RoboDK station: 로봇팔 이동.rdk

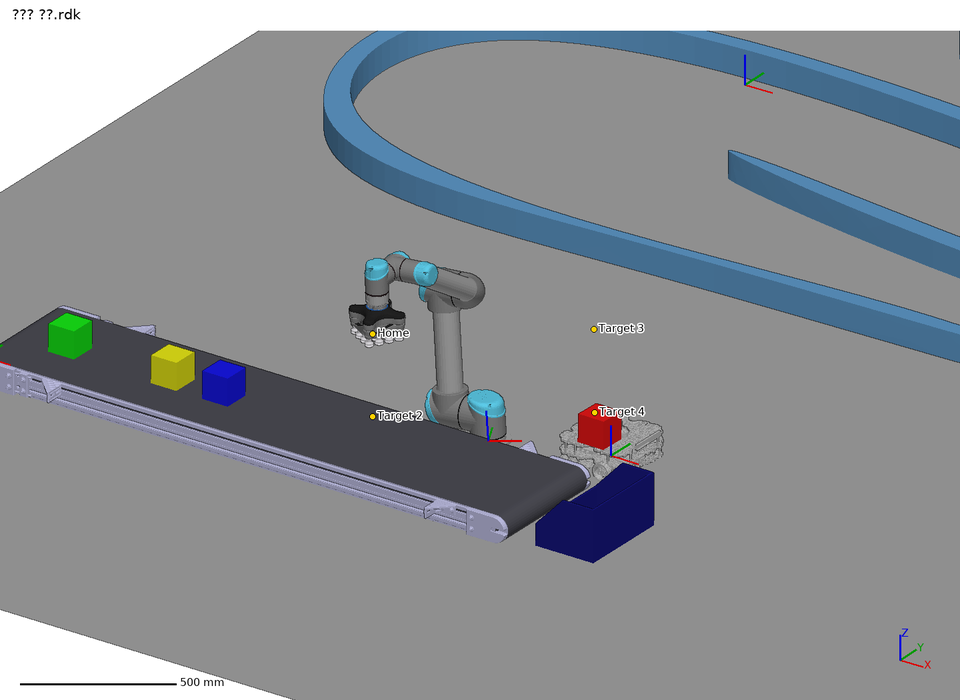
[picture v0: the station drawn from its stored meshes, robots at their saved joint values, targets as dots, program paths as lines]
Station 로봇팔 이동 (saved by RoboDK 5.7.4). Poses are relative to the parent item; angles as X-Y-Z fixed-axis rotations.
Station parameters (name, value as stored): LOAD_READY, 1
  - frame MainFrame at (0, 0, 0) mm
    - target Home (Cartesian target) at (651.26, -3006.26, 497.49) mm, rotated rx -179.45 ry 0.15 rz -30.37 deg; joints [-119.255, -87.831, -60.137, -122.512, 86.049, -150.839] of UR5
    - target Target 2 (Cartesian target) at (637.94, -2986.86, 192) mm, rotated rx -178.43 ry 0.43 rz -30.31 deg; joints [-119.878, -81.815, -111.866, -77.787, 86.288, -151.442] of UR5
    - target Target 3 (Cartesian target) at (1212.52, -2572.15, 497.3) mm, rotated rx -179.45 ry 0.15 rz -30.37 deg; joints [-13.799, -91.747, -62.441, -119.492, 91.513, -45.448] of UR5
    - target Target 4 (Cartesian target) at (1213.24, -2569.51, 200.09) mm, rotated rx -179.45 ry 0.15 rz -30.37 deg; joints [-12.8, -86.409, -112.222, -75.023, 91.577, -44.451] of UR5
  - frame UR5 Base at (820, -2600, 0) mm, rotated rx -1.94 ry -3.6 rz 28.07 deg
    - robot UR5: 6 axes
        modified DH rows (alpha deg, a mm, theta deg, d mm): 0, 0, 0, 89.2; 90, 0, 180, 0; 0, 425, 0, 0; 0, 392, 0, 109.3; -90, 0, 0, 94.75; 90, 0, 180, 82.5
        joint limits [-360, -360, -360, -360, -360, -360] to [360, 360, 360, 360, 360, 360]; home [0, -90, -90, 0, 90, 0]; saved at [-114.958, -89.114, -59.218, -122.443, 86.096, -146.532]
      - tool OnRobot VG10 Vacuum Gripper, TCP at (-36.63, 0, 130.9) mm, size 145.4 x 145.4 x 118.3 mm
  - object Floor at (0, -3000, 0) mm, size 3000 x 3000 x 0 mm, geometry from Floor (1).sld
  - object Floor at (3000, -3000, 0) mm, size 3000 x 3000 x 0 mm, geometry from Floor (1).sld
  - object Floor at (0, 0, 0) mm, size 3000 x 3000 x 0 mm, geometry from Floor (1).sld
  - object Bin Red at (2930, 150, 0) mm, rotated rx 0 ry 0 rz -180 deg, size 225 x 337.5 x 191.2 mm, geometry from Bin-Red.sld
  - object Floor at (3000, 0, 0) mm, size 3000 x 3000 x 0 mm, geometry from Floor (1).sld
  - object Bin Blue at (1380, -2800, 0) mm, rotated rx 0 ry 0 rz -180 deg, size 225 x 337.5 x 191.2 mm, geometry from Bin-Blue.sld
  - object path at (5000, -200, 0) mm, size 3159.6 x 1446.5 x 100 mm, geometry from path.step
  - object path2 at (-2520, -560, 40) mm, rotated rx 0 ry 0 rz 180 deg, size 3159.6 x 1446.5 x 100 mm, geometry from path.step
  - frame Conveyor Belt (2m) Base at (-740, -3190, 100) mm
    - robot Conveyor Belt (2m): 1 axes
        modified DH rows (alpha deg, a mm, theta deg, d mm): 0, 0, 0, 0 linear
        base shift (0, 0, 0) mm, rotated rx 0 ry 90 rz 0 deg
        joint limits [-500000] to [500000]; home [0]; saved at [0]
    - object Blue at (800, 200, 0) mm, size 100 x 100 x 100 mm, geometry from Blue.step
    - object Yellow at (600, 200, 0) mm, size 100 x 100 x 100 mm, geometry from Yellow.step
    - object Green at (200, 200, 0) mm, size 100 x 100 x 100 mm, geometry from Green.step
  - frame turtlebot Base at (1224.75, -2495.03, 20) mm
    - object turtlebot3_waffle (1) at (0, 0, 0) mm, size 280.7 x 305.1 x 138.1 mm, geometry from turtlebot3_waffle (1).step
    - object Red at (10.09, -79.28, 88.06) mm, rotated rx -1.02 ry 0.28 rz -0.1 deg, size 100 x 100 x 100 mm, geometry from Red.step
  - Python program Prog1 (listed below)

--- Python program Prog1 ---
from robodk import robolink
import time

RDK = robolink.Robolink()

# =========================
# RoboDK 아이템 찾기
# =========================
robot = RDK.Item("UR5")
tool = RDK.Item("OnRobot VG10 Vacuum Gripper")
red_box = RDK.Item("Red")
turtle_base = RDK.Item("turtlebot Base")

home = RDK.Item("Home")
target2 = RDK.Item("Target 2")   # Pick 위치
target3 = RDK.Item("Target 3")   # 이동 중간 위치
target4 = RDK.Item("Target 4")   # Place 위치

def check(item, name):
    if not item.Valid():
        raise Exception(f"'{name}' 을 찾을 수 없습니다. 왼쪽 트리 이름을 확인하세요.")

check(robot, "UR5")
check(tool, "OnRobot VG10 Vacuum Gripper")
check(red_box, "Red")
check(turtle_base, "turtlebot Base")
check(home, "Home")
check(target2, "Target 2")
check(target3, "Target 3")
check(target4, "Target 4")

# 속도 조절
robot.setSpeed(100)

# =========================
# Pick & Place 동작
# =========================

print("1. Home 이동")
robot.MoveJ(home)

print("2. Pick 위치 Target 2 이동")
robot.MoveJ(target2)
time.sleep(0.5)

print("3. Red 흡착")
red_abs = red_box.PoseAbs()
red_box.setParentStatic(tool)
red_box.setPoseAbs(red_abs)
time.sleep(0.5)

print("4. Target 3 이동")
robot.MoveJ(target3)

print("5. Place 위치 Target 4 이동")
robot.MoveJ(target4)
time.sleep(0.5)

print("6. Red를 터틀봇 위에 놓기")
red_abs = red_box.PoseAbs()
red_box.setParentStatic(turtle_base)
red_box.setPoseAbs(red_abs)
time.sleep(0.5)

print("7. Target 3 복귀")
robot.MoveJ(target3)

print("8. Home 복귀")
robot.MoveJ(home)

# 터틀봇 출발 신호
RDK.setParam("LOAD_READY", "1")

print("Pick & Place 완료")
